// TIA Portal V19 export
VAR_GLOBAL   // PLC tag table "Default tag table"
   "C1.1_I" AT %I2.0 : Bool;
   "C1.2_I" AT %I2.1 : Bool;
   "C2.1_I" AT %I2.2 : Bool;
   "C2.2_I" AT %I2.3 : Bool;
   "C3.1_I" AT %I2.4 : Bool;
   "C3.2_I" AT %I2.5 : Bool;
   Fotocelle_I AT %I2.6 : Bool;
   A_IG_I AT %I3.1 : Bool;
   B_IG_I AT %I3.2 : Bool;
   Bryter_S1_Ved_HMI_I AT %I0.0 : Bool;
   Bryter_S5_Ved_HMI_I AT %I0.4 : Bool;
   Bryter_Høyre_Skap_I AT %I3.3 : Bool;
   Bryter_Venstre_Skap_I AT %I3.4 : Bool;
   Tag_10 AT %IW64 : Word;
   Bryter_S2_Ved_HMI_I AT %I0.1 : Bool;
   Bryter_3_Ved_HMI_I AT %I0.2 : Bool;
   Bryter_S4_Ved_HMI_I AT %I0.3 : Bool;
   Tag_2 AT %I3.0 : Bool;
   "A-IG" AT %I4.0 : Bool;
   "16cm_Nærhetsføler_ved_robot" AT %I5.5 : Bool;
   "8cm_Nærhetsføler_ved_robot" AT %I5.6 : Bool;
   Tag_7 AT %I5.7 : Bool;
   "12cm_Nærhetsføler_ved_robot" AT %I5.4 : Bool;
   "12_CM_Sluppet" AT %I5.1 : Bool;
   "8_CM_Sluppet" AT %I5.2 : Bool;
   "16_CM_Sluppet" AT %I5.3 : Bool;
   "16cm_knapp_main_skap" AT %I0.5 : Bool;
   "12cm_plukk_robot" AT %Q2.0 : Bool;
   "16cm_plukk_robot" AT %Q2.1 : Bool;
   "8_plukk_robot" AT %Q2.2 : Bool;
   V2 AT %Q3.1 : Bool;
   V1 AT %Q3.0 : Bool;
   Tag_14 AT %Q0.2 : Bool;
   V3 AT %Q3.2 : Bool;
   C3 AT %Q3.3 : Bool;
   Tag_9 AT %Q3.4 : Bool;
   Tag_11 AT %QW68 : Word;
   Tag_1 AT %QW70 : Word;
   V4_Utgang AT %Q4.0 : Bool;
   V5_Utgang AT %Q4.1 : Bool;
   V6_Utgang AT %Q4.2 : Bool;
   "C1.1_M" AT %M0.0 : Bool;
   "C1.2_M" AT %M0.1 : Bool;
   "C2.1_M" AT %M0.2 : Bool;
   "C2.2_M" AT %M0.3 : Bool;
   "C3.1_M" AT %M0.4 : Bool;
   "C3.2_M" AT %M0.5 : Bool;
   Fotocelle_M AT %M0.6 : Bool;
   A_IG_M AT %M0.7 : Bool;
   Bryter_Høyre_Skap_M AT %M1.1 : Bool;
   B_IG_M AT %M1.0 : Bool;
   Bryter_S1_Ved_HMI_M AT %M2.0 : Bool;
   Bryter_S2_Ved_HMI_M AT %M2.1 : Bool;
   Bryter_S3_Ved_HMI_M AT %M2.2 : Bool;
   System_Byte AT %MB8001 : Byte;
   FirstScan AT %M8001.0 : Bool;
   DiagStatusUpdate AT %M8001.1 : Bool;
   AlwaysTRUE AT %M8001.2 : Bool;
   AlwaysFALSE AT %M8001.3 : Bool;
   Clock_Byte AT %MB8000 : Byte;
   Clock_10Hz AT %M8000.0 : Bool;
   Clock_5Hz AT %M8000.1 : Bool;
   "Clock_2.5Hz" AT %M8000.2 : Bool;
   Clock_2Hz AT %M8000.3 : Bool;
   "Clock_1.25Hz" AT %M8000.4 : Bool;
   Clock_1Hz AT %M8000.5 : Bool;
   "Clock_0.625Hz" AT %M8000.6 : Bool;
   "Clock_0.5Hz" AT %M8000.7 : Bool;
   Kloss1_8cm AT %M10.0 : Bool;
   "delay_set_10.2" AT %M10.1 : Bool;
   Kloss2_8cm AT %M10.2 : Bool;
   Tag_8 AT %M20.1 : Bool;
   V1_Kloss1_U AT %M11.0 : Bool;
   V1_Kloss2_U AT %M11.1 : Bool;
   "delay_set_10.4" AT %M10.3 : Bool;
   Kloss3_8cm AT %M10.4 : Bool;
   V1_Kloss3_U AT %M11.2 : Bool;
   Kloss1_12cm AT %M12.0 : Bool;
   Kloss2_12cm AT %M12.2 : Bool;
   Kloss3_12cm AT %M12.4 : Bool;
   "delay_set_12.4" AT %M12.3 : Bool;
   "delay_set_12.2" AT %M12.1 : Bool;
   V2_Kloss2_U AT %M13.1 : Bool;
   V2_Kloss3_U AT %M13.2 : Bool;
   V2_Kloss1_U AT %M13.0 : Bool;
   Kloss4_12cm AT %M12.6 : Bool;
   "delay_set_12.6" AT %M12.5 : Bool;
   V2_Kloss4_U AT %M13.3 : Bool;
   "delay_set_14.2" AT %M14.1 : Bool;
   "delay_set_14.4" AT %M14.3 : Bool;
   "delay_set_14.6" AT %M14.5 : Bool;
   Kloss4_16cm AT %M14.6 : Bool;
   Kloss1_16cm AT %M14.0 : Bool;
   Kloss2_16cm AT %M14.2 : Bool;
   Kloss3_16cm AT %M14.4 : Bool;
   "delay_set_15.0" AT %M14.7 : Bool;
   Kloss5_16cm AT %M15.0 : Bool;
   V3_Kloss1_U AT %M15.1 : Bool;
   V3_Kloss2_U AT %M15.2 : Bool;
   V3_Kloss3_U AT %M15.3 : Bool;
   V3_Kloss4_U AT %M15.4 : Bool;
   V3_Kloss5_U AT %M15.5 : Bool;
   Bryter_Venstre_Skap_M AT %M1.2 : Bool;
   Bryter_S4_Ved_HMI_M AT %M2.3 : Bool;
   Bryter_S5_Ved_HMI_M AT %M2.4 : Bool;
   Ventil_4_UT AT %M50.0 : Bool;
   Ventil_5_UT AT %M50.1 : Bool;
   Ventil_6_UT AT %M50.2 : Bool;
   "16CM_Pall_Full" AT %M5.0 : Bool;
   "12CM_Pall_Full" AT %M5.1 : Bool;
   "8CM_Pall_Full" AT %M5.2 : Bool;
   Tag_15 AT %I3.5 : Bool;
   Hent_8cm_til_Servo_Q AT %Q6.0 : Bool;
   Hent_12cm_til_Servo_Q AT %Q6.1 : Bool;
   Hent_16cm_til_Servo_Q AT %Q6.2 : Bool;
   Lever_12cm_til_servo_Q AT %Q6.4 : Bool;
   Lever_8cm_til_servo_Q AT %Q6.5 : Bool;
   Lever_16cm_til_servo_Q AT %Q6.6 : Bool;
   Ved_HentPos8cm_fra_servo AT %I6.0 : Bool;
   Ved_hentPos12cm_fra_servo AT %I6.1 : Bool;
   Ved_hentPos16cm_fra_servo AT %I6.2 : Bool;
   C4_PlussPos_I AT %I4.1 : Bool;
   C4_MinPos_I AT %I4.2 : Bool;
   C5_PlussPos_I AT %I4.3 : Bool;
   C5_MinPos_I AT %I4.4 : Bool;
   C6_PlussPos_I AT %I4.5 : Bool;
   C6_MinPos_I AT %I4.6 : Bool;
   C4_Retur_Set AT %M51.0 : Bool;
   Tag_3 AT %M1000.0 : Bool;
   "8cm_Pall_På_Plass" AT %M52.0 : Bool;
   Bekreftet_levert_pall_16cm_fra_servo AT %I6.5 : Bool;
   Bekreftet_levering_8_cm_fra_servo AT %I6.3 : Bool;
   Vent_ny_pall_8cm AT %M52.1 : Bool;
   Vent_ny_pall_16cm AT %M60.0 : Bool;
   Tag_4 AT %I0.6 : Bool;
   "16cm_pall_på_plass" AT %M60.1 : Bool;
   C6_retur_set AT %M60.3 : Bool;
   tag AT %M60.2 : Bool;
END_VAR
